TYPE ExampleTableRow :
STRUCT
	Name : STRING;
	Value : INT;
END_STRUCT
END_TYPE

(* stored: Version 1.1.0.1, ProductVersion 3.1.4024.15
   DUT ExampleTableRow: Id {a5f4ef32-d089-4857-b5e2-277cda58097b} *)
